// TIA Portal V17 export
// export: Created 2022-07-20T07:02:30.0863308Z, ExportSetting WithDefaults, DisplayName Totally Integrated Automation Portal, DisplayVersion V17, DisplayName TIA Portal Openness, DisplayVersion V17, DisplayName TIA Portal Version Control Interface, DisplayVersion V17, DisplayName SINAMICS Startdrive Advanced, DisplayVersion V17, DisplayName SINAMICS Startdrive G130, G150, S120, S150, SINAMICS MV, S210, DisplayVersion V17, DisplayName SINAMICS Startdrive G110M, G120, G120C, G120D, G120P, G115D, DisplayVersion V17, DisplayName STEP 7 Professional, DisplayVersion V17, DisplayName STEP 7 Safety, DisplayVersion V17, DisplayName WinCC Advanced, DisplayVersion V17
DATA_BLOCK "LAcycCom_RequestBuffer"   // DB30500
TITLE = LAcycCom_RequestBuffer
{ S7_Optimized_Access := 'TRUE' }
AUTHOR : APC_ERLF
FAMILY : AcycCom
VERSION : 1.1
// Support: tech.team.motioncontrol@siemens.com 
// Fax: +49 (0) 9131/98-1297
// stored: AutoNumber true, DBAccessibleFromOPCUA true, DBAccessibleFromWebserver true, InstanceOfName LAcycCom_typeRequestBuffer, InstanceOfType UDT, IsOnlyStoredInLoadMemory false, IsWriteProtectedInAS false
"LAcycCom_typeRequestBuffer"
   // VAR
   //    header { ExternalWritable := 'False'; S7_SetPoint := 'True'} : "LAcycCom_typeRequestBufferHeader";
   //    elements { ExternalWritable := 'False'; S7_SetPoint := 'True'} : Array[0.."LACYCCOM_BUFFER_ELEMENTS_UPPER_LIM"] of "LAcycCom_typeRequestBufferElement";
   // END_VAR
BEGIN
END_DATA_BLOCK
